PROGRAM PRG_Alt
VAR
	test : REAL;
	PT : REAL := 50.5;
	TT : REAL := 11.5;
	SV : BOOL;
END_VAR

END_PROGRAM

(* stored: Version 1.1.0.1
   POU PRG_Alt: Id {c9677053-391b-466b-b0c6-a03af7227cd2}, SpecialFunc None *)
